RoboDK station: RK3 extrudy.rdk

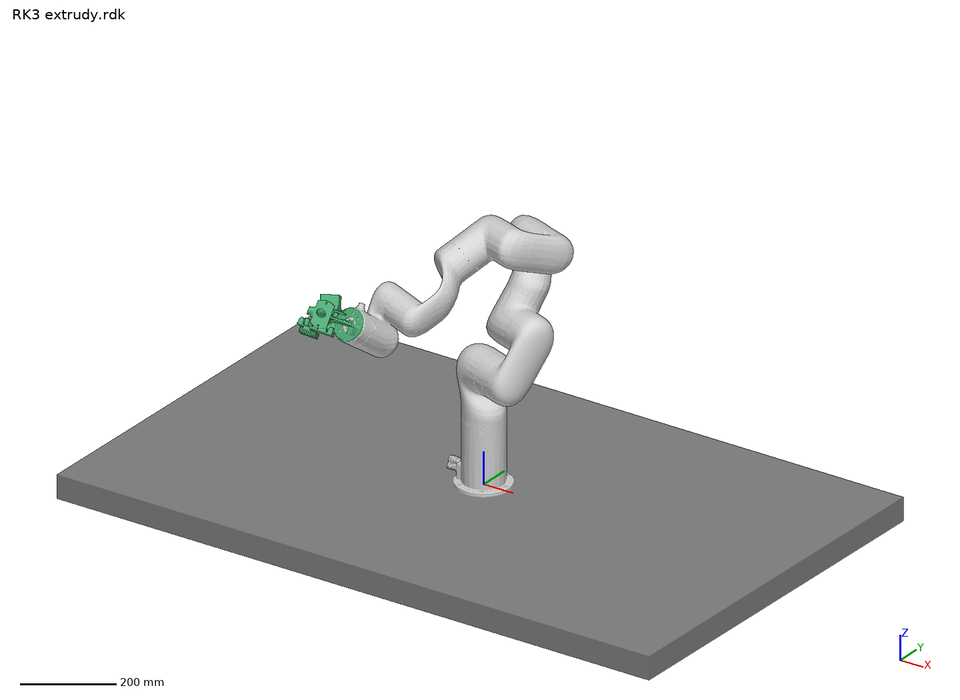
[picture v0: the station drawn from its stored meshes, robots at their saved joint values, targets as dots, program paths as lines]
Station RK3 extrudy (saved by RoboDK 5.5.0). Poses are relative to the parent item; angles as X-Y-Z fixed-axis rotations.
  - frame uFactory xArm6 Base at (0, 0, 0) mm
    - robot uFactory xArm6: 6 axes, payload 5 kg, reach 632 mm, repeatability 0.1 mm, weight 9.5 kg
        modified DH rows (alpha deg, a mm, theta deg, d mm): 0, 0, 0, 267; -90, 0, -79.35, 0; 0, 289.489, 79.35, 0; -90, 77.5, 0, 342.5; 90, 0, 0, 0; -90, 76, 0, 97
        joint limits [-360, -118, -225, -360, -97, -360] to [360, 120, 11, 360, 180, 360]; home [0, 0, 0, 0, 0, 0]; saved at [-109.558, -36.068, -32.133, 170.933, 57.51, -73.802]
      - tool WASP extruder, TCP at (0, 0, 107) mm, rotated rx 0 ry -30 rz 0 deg, size 160.2 x 105.1 x 183.1 mm, geometry from extruderModel2.stp
    - object table at (0, 0, 0) mm, rotated rx 90 ry 0 rz 0 deg, size 1500 x 55 x 920 mm, geometry from table.obj
  - machining project Print3D settings: rotZ(0) | rotX(0)*rotY(0) | rotz(0) | onStart | onPathStart | onApproach | onPoint | onRetract | onFinish | SetRPM(%1) | SetTool(%1) | Prog1 | default | default | OutOnMov(%1) | OutOffMov(%1) | onPathFinish | M_RunCode(%1)
  - Python program modbus_extruder (listed below)

--- Python program modbus_extruder ---
# Type help("robodk.robolink") or help("robodk.robomath") for more information
# Press F5 to run the script
# Documentation: https://robodk.com/doc/en/RoboDK-API.html
# Reference:     https://robodk.com/doc/en/PythonAPI/robodk.html
# Note: It is not required to keep a copy of this file, your Python script is saved with your RDK project
#!/usr/bin/env python3
# Software License Agreement (BSD License)
#
# Copyright (c) 2020, UFACTORY, Inc.
# All rights reserved.
#
# Author: Vinman <vinman.wen@ufactory.cc> <vinman.cub@gmail.com> and Chris

"""
Control the WASP extruder assembly through Modbus protocol
"""

import os
import sys
import time
sys.path.append(os.path.join(os.path.dirname(__file__), '../xArm-Python-SDK-master'))

#receive variables from RoboDK
move = RDK.getParam('move')
from xarm.wrapper import xarm_api
from configparser import ConfigParser
parser = ConfigParser()
parser.read('../robot.conf')
try:
    ip = parser.get('xArm', 'ip')


arm = XArmAPI(ip)
time.sleep(0.5)
if arm.warn_code != 0:
    arm.clean_warn()
if arm.error_code != 0:
    arm.clean_error()

arm.motion_enable(True)
arm.set_mode(0)
arm.set_state(0)

code = arm.set_tgpio_modbus_timeout(20)
print('set_tgpio_modbus_timeout, code={}'.format(code))

# set tool gpio modbus baudrate
code = arm.set_tgpio_modbus_baudrate(115200)
print('set_tgpio_modbus_baudrate, code={}'.format(code))
time.sleep(1)


data_frame = [0x08, 0x10, 0x00, 0x01, 0x00, 0x03, 0x06, 0x00, (move), 0x00, (dir), 0x00, (speed)]
    ret = arm.core.tgpio_set_modbus(data_frame, len(data_frame)) #setup these variables as hex values

    time.sleep(2)
